// TwinCAT 3 PLC project Facade
// ProgramVersion: 3.1.4023.0
// libraries:
//   Tc2_Standard, * (Beckhoff Automation GmbH)
//   Tc2_System, * (Beckhoff Automation GmbH)
//   Tc3_Module, * (Beckhoff Automation GmbH)
// project tree:
//   / Class Diagram.TcCD (not stored), PlcTask.TcTTO
//   Classes/ FacadePrinterNormal.TcPOU, Printer.TcPOU
//   POUs/ MAIN.TcPOU, PrincipalClient.TcPOU, PrincipalClient2.TcPOU
// real-time tasks:
//   TASK PlcTask: cycle T#10ms, priority 20, ADS port 350

CONFIGURATION Facade
    RESOURCE PLC ON TwinCAT3
        TASK PlcTask(INTERVAL := T#10ms, PRIORITY := 20);
        PROGRAM MAIN WITH PlcTask : MAIN;
    END_RESOURCE
END_CONFIGURATION

// ---- POUs/MAIN.TcPOU
PROGRAM MAIN
VAR
END_VAR

PrincipalClient();
PrincipalClient2();

END_PROGRAM

// ---- POUs/PrincipalClient.TcPOU
PROGRAM PrincipalClient
VAR
	i1 : Printer;	
	i2 : Printer;
	i3 : Printer;
	
	startdemo : BOOL;
END_VAR

//Se trata de una ejemplo sencillo que imprime documentos en uno u otro formato. 
//El código nos ayudará a entender mejor su funcionamiento.

//This is a simple example that prints documents in one format or another.
//The code will help us better understand how it works.

(*
Como podemos ver la clase cliente se encarga de invocar a la impresora, y configurarla para después imprimir varios documentos .
Ahora bien prácticamente todos los documentos que escribimos tienen la misma estructura (formato A4, Color , PDF). Estamos continuamente repitiendo código. 
Vamos a construir una nueva clase FachadaImpresoraNormal que simplifique la impresión de documentos que sean los más habituales.
*)

IF  startdemo THEN
	
	startdemo := FALSE;
	
	i1.setSheet('a1');
  	i1.setColor(TRUE);
  	i1.setdocumentType('pdf');
  	i1.setText('text 1');
  	i1.printDocument();
  	 
  	
  	i2.setSheet('a2');
  	i2.setColor(FALSE);
  	i2.setdocumentType('rtf');
  	i2.setText('text 2');
  	i2.printDocument();
  	 
  	
  	i3.setSheet('a3');
  	i3.setColor(TRUE);
  	i3.setdocumentType('excel');
  	i3.setText('text 3');
  	i3.printDocument();	
END_IF

END_PROGRAM

// ---- Classes/Printer.TcPOU
FUNCTION_BLOCK PUBLIC Printer
VAR
	 documentType: STRING ;
     sheet: STRING ;
     color : BOOL ;
     text: STRING ;
END_VAR

PROPERTY PUBLIC getDocumentType : STRING
GET
getDocumentType := documentType;
END_GET
END_PROPERTY

PROPERTY PUBLIC getSheet : STRING
GET
getSheet := sheet;
END_GET
END_PROPERTY

PROPERTY PUBLIC getText : STRING
GET
getText := text;
END_GET
END_PROPERTY

PROPERTY PUBLIC isColor : BOOL
GET
isColor := color;
END_GET
END_PROPERTY

METHOD PUBLIC printDocument
VAR
	stext1 : STRING;
	stext2 : STRING;
	stext3 : STRING;
	stext4 : STRING;
	stext : STRING;
	strSFCErrorStep : STRING:='';
END_VAR
//    System.out.println("printing:"+ text+ ",color:"
//        + color+",type:"+DocumentType+",sheet :"+sheet);
		
stext1 := CONCAT(STR1:='printing: ' , STR2:= text);
stext2 := CONCAT(STR1:=', color: ' , STR2:= TO_STRING(color));
stext3 := CONCAT(STR1:=', type: ' , STR2:= DocumentType);
stext4 := CONCAT(STR1:=', sheet: ' , STR2:= sheet);
stext :=  CONCAT(STR1:=stext1 , STR2:=CONCAT(STR1:=stext2 , STR2:=CONCAT(STR1:=stext3 , STR2:=stext4)));
		
 ADSLOGSTR( msgCtrlMask := ADSLOG_MSGTYPE_LOG, msgFmtStr := stext, strArg := strSFCErrorStep);
END_METHOD

METHOD PUBLIC setColor
VAR_INPUT
	color : BOOL;
END_VAR
THIS^.color := color;
END_METHOD

METHOD PUBLIC setDocumentType
VAR_INPUT
	documentType :STRING;
END_VAR
THIS^.documentType := documentType;
END_METHOD

METHOD PUBLIC setSheet
VAR_INPUT
	sheet: STRING ;
END_VAR
THIS^.sheet := sheet;
END_METHOD

METHOD PUBLIC setText
VAR_INPUT
	text :STRING ;
END_VAR
THIS^.text := text;
END_METHOD

END_FUNCTION_BLOCK

// ---- POUs/PrincipalClient2.TcPOU
PROGRAM PrincipalClient2
VAR
	facade1 : FacadePrinterNormal(text:= 'text 1', color:= TRUE , sheet:= 'A1', documentType:='PDF');
         
    facade2 : FacadePrinterNormal(text:= 'text 2', color:= FALSE , sheet:= 'A2', documentType:='Excel');
	                  
    i3 : printer;
	
	startdemo : BOOL;
	
END_VAR


IF  startdemo THEN
	
	startdemo := FALSE;

	facade1.print();
			
	facade2.print();
			 
	i3.setSheet('A3');
    i3.setColor(TRUE);
    i3.setDocumenttype('RTF');
    i3.setText('text 3');
    i3.printDocument();
	
END_IF

END_PROGRAM

// ---- Classes/FacadePrinterNormal.TcPOU
FUNCTION_BLOCK PUBLIC FacadePrinterNormal
VAR_INPUT
END_VAR
VAR_OUTPUT
END_VAR
VAR
	printer :  Printer;
END_VAR

METHOD FB_init : BOOL
VAR_INPUT
	bInitRetains : BOOL; // if TRUE, the retain variables are initialized (warm start / cold start)
	bInCopyCode : BOOL;  // if TRUE, the instance afterwards gets moved into the copy code (online change)
	text : STRING;
	color : BOOL;
	sheet : STRING;
	documentType : STRING;
	
END_VAR

printer.setColor(color);
printer.setSheet(sheet);
printer.setdocumentType(documentType);
printer.setText(text);
END_METHOD

METHOD print
printer.printDocument();
END_METHOD

END_FUNCTION_BLOCK
